// TIA Portal V20 export
DATA_BLOCK "R_TRIG_DB"   // DB13
// stored: InstanceOfName R_TRIG, OfSystemLibElement R_TRIG, OfSystemLibVersion 1.0
"R_TRIG"
   // VAR_INPUT
   //    CLK : Bool;
   // END_VAR
   // VAR_OUTPUT
   //    Q : Bool;
   // END_VAR
   // VAR
   //    Stat_Bit : Bool;
   // END_VAR
BEGIN
END_DATA_BLOCK
